Fanuc KAREL source: MP0115.KL

-- PROVISIONAL review KL for V770-1; original PC SHA256 2a7ccc4ed1a0243602ee84b997f0a4b7691ae1d058b638e73d01dd0becbb22e3
-- Incomplete behavior may be omitted. Consult companion uncertainty JSON. Do not deploy.
PROGRAM MP0115
%NOLOCKGROUP
-- UNRESOLVED_LOCAL_POOL 8 cells at code offset 61; source declarations unknown
-- DIRECT_LOCAL_WORD_ACCESS alone does not prove INTEGER, REAL, or BOOLEAN
BEGIN
  -- UNRESOLVED_PC offsets 0-1; opcodes 7B
  -- UNRESOLVED_PC offsets 6-18; opcodes 2D,9D,52,7F
  -- UNRESOLVED_PC offsets 23-28; opcodes 7F,7B
  -- UNRESOLVED_PC offsets 33-49; opcodes 2D,2E,69,7F
  -- UNRESOLVED_PC offsets 54-66; opcodes 7F,2B,2C,7B
  -- UNRESOLVED_PC offsets 71-82; opcodes 2E,23
  -- UNRESOLVED_PC offsets 87-98; opcodes 2E,23
  -- UNRESOLVED_PC offsets 103-114; opcodes 2E,23
  -- UNRESOLVED_PC offsets 119-130; opcodes 2E,23
  -- UNRESOLVED_PC offsets 135-146; opcodes 2E,23
  -- UNRESOLVED_PC offsets 151-162; opcodes 2E,23
  -- UNRESOLVED_PC offsets 167-193; opcodes 21,21,21,54,52,23
  -- UNRESOLVED_PC offsets 198-202; opcodes 7F
  -- UNRESOLVED_PC offsets 207-223; opcodes 27,27,2E,27,2E,AA
  -- UNRESOLVED_PC offsets 228-232; opcodes 7F
END MP0115
